FUNCTION_BLOCK FB_HTTP_Get_Elpris
VAR_INPUT
	bSend			: BOOL;
	timDataMomentan:REFERENCE TO ST_timData;
	timData: REFERENCE TO ARRAY[0..87600] OF ST_timData;
	stringDatumTid: STRING;
	timIndex: REFERENCE TO INT;
END_VAR
VAR_IN_OUT
	fbClient			: FB_IotHttpClient;
END_VAR
VAR_OUTPUT
	bBusy				: BOOL;
	bError				: BOOL;
END_VAR
VAR
		elpriserTimme: ARRAY[0..23] OF ST_elpriserTimme; //från elpriserjustnu.se
	fbRequest			: FB_IotHttpRequest;

	fbJson				: FB_JsonDomParser;
	
		fbJsonDataType	: FB_JsonReadWriteDataType;
		felkod			: HRESULT;			
	pContent: PVOID;
	nState				: UDINT;
	RisingEdge			: R_TRIG;
	
	bGetContentResult	: BOOL;
	sContent			: STRING(5000);
	
	bGetJsonResult		: BOOL;
	jsonDoc				: SJsonValue;
	jsonVal				: SJsonValue;
	sResultValue		: STRING;
	
	nReqCount			: UDINT;	
	nResCount			: UDINT;
	nValidResCount		: UDINT;
	nErrCount			: UDINT;
	Vaerde: LINT;
	Energi: REAL;
	Energilaegsta: REAL :=100000.0 ;
	Energihoegsta: REAL;
	n: INT;
	Funkar: BOOL;
	nisse: INT;
	kod1: UINT;
	kod2: UINT;
	Location: STRING(200);
	
	
	storlek: UINT;
	storleken: UDINT;
	nIndex: UDINT;
	nSize: UDINT;
	sJsonArrayIndex: Sjsonvalue;
	
	sJsonArray			:SJsonValue;

	SCopiedJson: STRING(200);

	
	sUri: STRING(255);
	stringDatum: STRING(255);
	stringAar: STRING(255);
	i: INT;
	nisses: REAL;
	kalle: INT;
	sldg: REAL;
	bTestRef1: BOOL;
END_VAR

RisingEdge(CLK:= bSend );


CASE nState OF
0:	
	IF RisingEdge.Q THEN 
	kalle:=kalle+1;
		 
			stringAar:=MID(stringDatumTid, 4, 4);
				stringDatum:=MID(stringDatumTid, 5, 9);
			 
			 sUri:=concat('/api/v1/prices/', stringAar);
			 sUri:=concat(sUri,'/'); 
			 sUri:=concat(sUri,stringDatum);
			 sUri:=concat(sUri,'_SE4.json');
			 //sUri:='/api/v1/prices/2023/02-14_SE4.json'

		IF fbRequest.SendRequest(sUri:=sUri, fbClient:=fbClient, eRequestType:=ETcIotHttpRequestType.HTTP_GET, 0, 0, 0) THEN
			
			nState:= 1;
			nReqCount:= nReqCount+1;
			bBusy:= TRUE;
			bError:= FALSE;
			sUri:='';
		END_IF					
	END_IF
1:
	IF NOT fbRequest.bBusy THEN
		nisse:=nisse+1;
			fbRequest.GetHeaderField(sField:='Location',pValue:=ADR(Location),nValueSize:= SIZEOF(Location));
		kod1:=fbRequest.nStatusCode;
		bError:= TRUE;
		IF NOT fbRequest.bError THEN	
			//Hämta data och lägg i string
		
		
		
			bGetContentResult:= fbRequest.GetContent(pContent:= ADR(sContent), nContentSize:= SIZEOF(sContent), bSetNullTermination:= TRUE);
		
			storleken:=fbRequest.nContentSize;
			
			IF fbRequest.nStatusCode >= 200 AND fbRequest.nStatusCode < 300 THEN
				bGetJsonResult:= FALSE;
				jsonDoc:= fbRequest.GetJsonDomContent(fbJson);
				IF jsonDoc <> 0 THEN
					bGetJsonResult:= TRUE;
					
					//sJsonArray:=fbJson.FindMember(jsonDoc, 'timeSeries');
				
					nSize:= LIMIT(1, fbJson.GetArraySize(jsonDoc), 100);
					
					FOR nIndex:= 0 TO (nSize-1) DO   //Alltid 0-23 timmar
						
						sJsonArrayIndex:= fbJson.GetArrayValueByIdx(jsonDoc, nIndex);
						
						fbJson.CopyJson(sJsonArrayIndex, SCopiedJson, SIZEOF(SCopiedJson));
						
						fbJsonDataType.SetSymbolFromJson(sCopiedJson, 'ST_elpriserTimme', SIZEOF(elpriserTimme[nIndex]), ADR(elpriserTimme[nIndex]));
												
					END_FOR
				
			(*	
				//Kopiera hela den importerade JSON-formaterade datasträngen och lägg i en motsvarande TwinCAT-struktur
				IF fbJsonDataType.SetSymbolFromJson(sContent, 'ST_elpriserJustNu24Timmar', SIZEOF(elpriserTimme), ADR(elpriserTimme), hrErrorCode=> felkod) THEN
						bError:= FALSE;
				END_IF	
		*)
		
		//Stoppa in dygnets elpriser

		
FOR i:= 0 TO (23) DO
	timData[timIndex+i].timPris:= elpriserTimme[i].SEK_per_kWh;
	//sldg:= elpriserTimme[i].SEK_per_kWh;
END_FOR

				nResCount:= nResCount+1 ;	
				

			END_IF
		END_IF
		nState:= 0;
		bBusy:= FALSE;
		IF bError THEN
			nErrCount:= nErrCount+1;
		END_IF
	END_IF  
END_IF	


END_CASE

END_FUNCTION_BLOCK

(* stored: Version 1.1.0.1, ProductVersion 3.1.4024.12
   POU FB_HTTP_Get_Elpris: Id {f266cfe8-b744-4fee-93c9-afadbb6020cc}, SpecialFunc None *)
